TYPE TankCtrl_Ctx :
STRUCT
	io		: TankCtrl_Io;
	hmi		: TankCtrl_Hmi;
	priv	: TankCtrl_Priv;
	state	: TankCtrl_States;
END_STRUCT
END_TYPE

(* stored: Version 1.1.0.1
   DUT TankCtrl_Ctx: Id {3a4f68d0-90bc-4071-8cc7-0cac0d1f240d} *)
